FUNCTION_BLOCK RobotA21_methods_backup EXTENDS KukaRobot
VAR_INPUT
	out8 : INT;
END_VAR
VAR_OUTPUT
	//forceStop AT %Q* : BOOL;
	//resetSignal AT %Q* : BOOL;
	
	//outputs AT %Q* : ARRAY[1..50] OF INT;
	//inputs AT %I* : ARRAY[1..20] OF INT;
	
	taskID : INT;
	completedTask : INT;
	(*
	operational : BOOL;
	reserved : BOOL;
	reservation : SectionEnum := SectionEnum.NULL_SECTION;
	tool : SectionEnum := SectionEnum.WOOD_BUNK;
	
	error : BOOL;
	errId : DINT;
	*)
END_VAR

taskID := outputs[1];
completedTask := inputs[1];

outputs[8].15 := 
	NOT strapper.enable AND 
	NOT strapper.execute;

outputs[8] := out8;

//{attribute 'monitoring' := 'variable'}
{attribute 'monitoring' := 'call'}
PROPERTY Busy : BOOL
GET
VAR
	//emptyOutput : ARRAY[1..50] OF INT;
END_VAR
//Busy stays TRUE until outputs are cleared AND completed task has elapsed
//Ready is always inverse of Busy
updateStatus();

Busy := taskID <> 0 OR completedTask <> 0;
END_GET
END_PROPERTY

METHOD commandEx : BOOL
VAR_INPUT
	newOutputs : REFERENCE TO ARRAY[1..50] OF INT;
END_VAR
//IF NOT Busy THEN
	//RETURN;
//END_IF

outputs := newOutputs;
commandEx := Done;

(*
CASE step OF
	SEND_COMMAND: //wait 1 cycle
		outputs := newOutputs;
		step := WAIT;
		
	WAIT:
		IF done THEN
			(*	
			IF NOT reset() THEN
				RETURN;
			END_IF
			
			step := 0;
			*)
			setCommandAndWait := TRUE;
		END_IF
		
END_CASE
*)
END_METHOD

//{attribute 'monitoring' := 'variable'}
{attribute 'monitoring' := 'call'}
PROPERTY Done : BOOL
GET
updateStatus();

Done :=
	completedTask = taskID AND
	taskID <> 0 AND
	completedTask <> 0;
END_GET
END_PROPERTY

METHOD eStop : BOOL
VAR_INPUT
END_VAR
//forceStop := TRUE;
//eStop := TRUE;
END_METHOD

METHOD idleCommand : BOOL
VAR_INPUT
END_VAR
MEMSET(ADR(outputs), 0, SIZEOF(outputs));
END_METHOD

//{attribute 'monitoring' := 'variable'}
{attribute 'monitoring' := 'call'}
PROPERTY Ready : BOOL
GET
updateStatus();

Ready := taskID = 0 AND completedTask = 0;
END_GET
END_PROPERTY

METHOD release : BOOL
VAR_INPUT
	sectionReservation : SectionEnum;
END_VAR
IF reservation = sectionReservation AND reserved THEN
	reservation := SectionEnum.NULL_SECTION;
	reserved := FALSE;
	release := TRUE;
END_IF
END_METHOD

METHOD reserve : BOOL
VAR_INPUT
	reserveRequest : SectionEnum;
END_VAR
(*
this method exists because chipboard and wood bunk operations use the same robot
both sections need to check if the robot is open to commands before use
*)
IF reserved AND reservation = reserveRequest THEN
	reserve := TRUE;

ELSIF (NOT reserved) AND reservation = SectionEnum.NULL_SECTION THEN
	reservation := reserveRequest;
	reserved := TRUE;
	reserve := TRUE;

END_IF
END_METHOD

METHOD reset : BOOL
//resetSignal := TRUE;
//done := FALSE;

MEMSET(ADR(outputs), 0, SIZEOF(outputs));
(*
IF ready AND completedTask = 0 THEN
	resetSignal := FALSE;
	reset := TRUE;
END_IF
*)
END_METHOD

METHOD resume : BOOL
VAR_INPUT
END_VAR
//forceStop := FALSE;

resume := NOT error AND errId = 0;
END_METHOD

METHOD updateStatus : BOOL
VAR_INPUT
END_VAR
taskID := outputs[1];
completedTask := inputs[1];
END_METHOD

END_FUNCTION_BLOCK

(* stored: Version 1.1.0.1, ProductVersion 3.1.4024.11
   POU RobotA21_methods_backup: Id {efb9e82d-b439-4af4-83dd-650c783cf15a}, SpecialFunc None
   Folder Properties: Id {1470e281-74ec-4518-8098-79ea9102a8ce}
   Property Busy: Id {36f726c9-efaa-434a-a1c8-56486f4162fa}
   Get Get: Id {5906f38f-d0d2-4d2d-8be6-88ced41b4f3b}
   Method commandEx: Id {8fc3402d-842f-49b2-a742-8eb20dbfc62e}
   Property Done: Id {ab94ac1b-392d-4717-865a-c69d3ca1ac59}
   Get Get: Id {28916bb1-7370-435c-8645-47a4a83c71f2}
   Method eStop: Id {e1024b7f-c1d4-4d1c-9f46-317992db8f6f}
   Method idleCommand: Id {cb7fdee8-9138-42c4-8337-08882bb01546}
   Property Ready: Id {4c2d0524-ba1a-4958-9001-5c4271371a41}
   Get Get: Id {fddc9d66-5ac0-4874-b9bf-99bf801e7b49}
   Method release: Id {182de378-6f51-4baf-ae92-3cea30133752}
   Method reserve: Id {3c30ee0c-30d5-4cc7-a478-76c2033cbe44}
   Method reset: Id {a996abf0-3a85-418d-8e1d-92f5d62c2de6}
   Method resume: Id {25c71382-5780-44f4-b01c-90131fe3f7f8}
   Method updateStatus: Id {1838f0e4-fc01-4a97-bf78-7907501315ae} *)
